// _750_8212_PFC200/Application/Utils/MATH_LinearInterpolation
FUNCTION MATH_LinearInterpolation : REAL
VAR_INPUT
	X : REAL;
	X1 : REAL;
	Y1 : REAL;
	X2 : REAL;
	Y2 : REAL;
END_VAR
VAR
END_VAR

IF Y1 <> Y2 THEN
	MATH_LinearInterpolation := Y1 + (X - X1) * ((Y2 - Y1)/(X2 - X1));
ELSE
	MATH_LinearInterpolation := Y1;
END_IF

END_FUNCTION

// _750_8212_PFC200/Application/ALGO/SOC/SOC
FUNCTION_BLOCK SOC
VAR_INPUT
	SOC : REFERENCE TO typSOC;
	StringMinMax : REFERENCE TO StringMinMax;
END_VAR
VAR_OUTPUT
END_VAR
VAR
	m_PreviousTime : TIME;
END_VAR

METHOD Calculate
VAR_INPUT
	SocValues : REFERENCE TO typSOC;
	//CellsValues : REFERENCE TO typCELLS_VALUES;
	StringMinMax : REFERENCE TO typMIN_MAX;
	StringCurrent : REAL;
END_VAR
VAR
	m_DeltaTime : LTIME;
	m_DeltaSOC : REAL;
END_VAR
IF (NOT __ISVALIDREF(SocValues)) THEN RETURN; END_IF;

IF (gvBMS.Fb_String.GetStringState() = eBMS_CURRENT_FLOW_STATE.AT_REST) THEN
	RecalibrateViaLookUpTable(SOC := SocValues, StringMinMax := StringMinMax);
ELSE
	m_DeltaTime := LTIME() - m_PreviousTime; m_PreviousTime := LTIME(); 	
	
	IF TO_LREAL(m_DeltaTime) > 0 THEN
		m_DeltaSOC := ((StringCurrent * TO_LREAL(m_DeltaTime))/STRING_CONFIG.SOC_STRING_CAPACITY_mAs) * 100 / 1000;
	END_IF
	
	SocValues.averageSOC_pct := SocValues.averageSOC_pct - m_DeltaSOC;
	SocValues.minimumSOC_pct := SocValues.minimumSOC_pct - m_DeltaSOC;
	SocValues.maximumSOC_pct := SocValues.maximumSOC_pct - m_DeltaSOC;
	
	CheckSOCLimits(SOC.SOC);
	
END_IF
END_METHOD

METHOD CheckSOCLimits
VAR_INPUT
	SOC : REFERENCE TO typSOC;
END_VAR
IF SOC.maximumSOC_pct > STRING_CONFIG.SOC_MAXIMUM_SOC THEN
	SOC.maximumSOC_pct := STRING_CONFIG.SOC_MAXIMUM_SOC;
END_IF

IF SOC.maximumSOC_pct < STRING_CONFIG.SOC_MINIMUM_SOC THEN
	SOC.maximumSOC_pct := STRING_CONFIG.SOC_MINIMUM_SOC;
END_IF

IF SOC.averageSOC_pct > STRING_CONFIG.SOC_MAXIMUM_SOC THEN
	SOC.averageSOC_pct := STRING_CONFIG.SOC_MAXIMUM_SOC;
END_IF

IF SOC.averageSOC_pct < STRING_CONFIG.SOC_MINIMUM_SOC THEN
	SOC.averageSOC_pct := STRING_CONFIG.SOC_MINIMUM_SOC;
END_IF

IF SOC.minimumSOC_pct > STRING_CONFIG.SOC_MAXIMUM_SOC THEN
	SOC.minimumSOC_pct := STRING_CONFIG.SOC_MAXIMUM_SOC;
END_IF

IF SOC.minimumSOC_pct < STRING_CONFIG.SOC_MINIMUM_SOC THEN
	SOC.minimumSOC_pct := STRING_CONFIG.SOC_MINIMUM_SOC;
END_IF
END_METHOD

METHOD GetSOCFromCharge : REAL
VAR_INPUT
	charge_As : REAL;
END_VAR
VAR
	charge_mAs : REAL;
END_VAR
VAR CONSTANT
	FACTOR_1000 : REAL := 10000;
END_VAR
charge_mAs := charge_As / FACTOR_1000;
GetSOCFromCharge := FACTOR_1000 * (charge_mAs/STRING_CONFIG.SOC_STRING_CAPACITY_mAs);
END_METHOD

METHOD RecalibrateViaLookUpTable
VAR_INPUT
	SOC : REFERENCE TO typSOC;
	StringMinMax : REFERENCE TO typMIN_MAX;
END_VAR
VAR
END_VAR

SOC.minimumSOC_pct := GetSOCFromVoltage(voltage_mV := StringMinMax.minimumCellVoltage_mV);
SOC.averageSOC_pct := GetSOCFromVoltage(voltage_mV := StringMinMax.averageCellVoltage_mV);
SOC.maximumSOC_pct := GetSOCFromVoltage(voltage_mV := StringMinMax.maximumCellVoltage_mV);
END_METHOD

END_FUNCTION_BLOCK

// _750_8212_PFC200/Application/CANBUS/CAN_TxCurrentSensor
FUNCTION_BLOCK CAN_TxCurrentSensor
VAR_INPUT
	ICanQueue : ICAN_Queue;
END_VAR
VAR_OUTPUT
END_VAR
VAR
	message : typCAN_SIGNAL_TX;
	test : BYTE;
	SendPeriod : Standard.TON;
END_VAR


SendPeriod(IN := NOT SendPeriod.Q, PT := T#100MS);

message.Data[1] := test;

IF NOT ICanQueue.isFull() THEN
	IF SendPeriod.Q THEN
		message.CAN_ID := 16#FF50;
		ICanQueue.addToQueue(message);
	END_IF
END_IF

END_FUNCTION_BLOCK

// _750_8212_PFC200/Application/Utils/Sigmoid
FUNCTION Sigmoid : REAL
VAR_INPUT
	X : REAL;
END_VAR


(*
version 1.2	10. mar. 2009
programmer 	hugo
tested by		tobias

this function calculates the sigmoid function

*)

IF X > 20.0 THEN
	Sigmoid := 1.0;
ELSIF x < -85.0 THEN
	Sigmoid := 0.0;
ELSE
	Sigmoid := 1.0 / (1.0 + EXP(-X));
END_IF;


(* revision history
hm	10.12.2007		rev 1.0
	original version

hm	11. mar. 2008		rev 1.1
	extended range of valid inputs to +inv / -inv

hm 10. mar. 2009		rev 1.2
	real constants updated to new systax using dot																																																																																																																																																																																																																																																																																																																																																																																																																																																																																																																																																																																																																																																																																																																																																																																																																																																																																																																																																																																																																																																											

*)

END_FUNCTION

// _750_8212_PFC200/Application/ALGO/StateEstimation/StateEstimation
FUNCTION_BLOCK StateEstimation
VAR_INPUT
END_VAR
VAR_OUTPUT
END_VAR
VAR
	m_SOC : SOC;
END_VAR

m_SOC.Calculate(SocValues := gvSOC.gvSOC, StringMinMax := gvBMS.gvMinMax, StringCurrent := 10);

END_FUNCTION_BLOCK

// _750_8212_PFC200/Application/CANBUS/CANUtils/CAN_TO_DINT
FUNCTION CAN_TO_DINT : DINT
VAR_INPUT
	StartByte : INT;
	Data : POINTER TO ARRAY[1..8] OF BYTE;
END_VAR
VAR
	b0 : BYTE;
    b1 : BYTE;
	b2 : BYTE;
    b3 : BYTE;
END_VAR

b0 := Data^[StartByte];
b1 := Data^[StartByte+1];
b2 := Data^[StartByte+2];
b3 := Data^[StartByte+3];

CAN_TO_DINT := TO_DINT(SHL(SHL(SHL(BYTE_TO_DWORD(b0), 8) OR BYTE_TO_DWORD(b1), 8) OR BYTE_TO_DWORD(b2), 8) OR BYTE_TO_DWORD(b3));

END_FUNCTION

// _750_8212_PFC200/Application/CANBUS/CANUtils/CAN_TO_REAL
FUNCTION CAN_TO_REAL : REAL
VAR_INPUT
	StartByte : INT;
	Data : POINTER TO ARRAY[1..8] OF BYTE;
	Offset : REAL := 0;
	Resolution : REAL := 0.1;
	PackMode : INT := 0; //0 - 2 bytes, 1 - 4 bytes
END_VAR
VAR
	b0 : BYTE;
	b1 : BYTE;
	b2 : BYTE;
	b3 : BYTE;
	_value : REAL;
	_iValue : INT;
	_diValue : DINT;
END_VAR

IF (Data = 0) THEN RETURN; END_IF;

CASE PackMode OF

0:

	_iValue := CAN_TO_INT(StartByte, Data);
	_value := TO_REAL(_iValue);
	
1:

	_diValue := CAN_TO_DINT(StartByte, Data);
	_value := TO_REAL(_diValue);
	
END_CASE;

CAN_TO_REAL := _value*Resolution + Offset;

END_FUNCTION
